VAR_GLOBAL CONSTANT
	cMAX_BLOCKED_SUP: INT := 3;
END_VAR

(* stored: Version 1.1.0.1, ProductVersion 3.1.0.19
   GVL Const_DRV: Id {30eb72f0-7a68-4c95-8647-0882641efcfa} *)
